Staubli VAL3: ReadProductName.pgx

public program ReadProductName(string x_sFileName (dimensions=1), bool& x_bRes (dimensions=1))
  local num l_nNum[3]
  local string l_sBuff
  local string l_sFileName
  local trsf l_trTrsf
begin

  //读取生产文件

  //参数初始化
  x_bRes=false
  l_sFileName=x_sFileName

  //判断文件是否存在
  if !$fileExists(l_sFileName)
    return
  endIf

  //关闭所有文件
  call FileDir:CloseAllFile()

  //文件是否可以打开
  nFileID=$fileOpen(l_sFileName,"r")
  if nFileID<0 or nFileID>9
    return
  endIf


  //读取每行并解析
  if $fileGet(nFileID,l_sBuff,1)!=1 or find(l_sBuff,"PRODUCT=")<0
    logMsg("读取产品名不正确")
    return
  else
    sProductName=right(l_sBuff,len(l_sBuff)-find(l_sBuff,"=")-1)
    logMsg("读取文件名："+sProductName)
    x_bRes=true
  endIf



end
